Fanuc KAREL source: kt00025.KL

PROGRAM KT00025
%STACKSIZE=65535
%PRIORITY=65535
%NOLOCKGROUP
VAR
I2 : INTEGER
OUT : INTEGER
-- UNRESOLVED DECLARATIONS (source type spelling not recovered)
-- H1 : ARRAY[2] OF TYPE_0x0017 (type_u16=0x2017)
BEGIN
-- UNRESOLVED_PC line 8 opcodes [2E 22 9D 33 B4] marker_code=0
I2=3
-- UNRESOLVED_PC line 10 opcodes [22 9D 33 B3 21 52 23] marker_code=35
END KT00025
